(* IEC 61131-3 sources: test/Class/HmiMapFile, 1 file *)

(* ---- HmiMapFile.st ---- *)
(*!
<Class
	Name               = "HmiMapFile"
	Revision           = "0.0"
	RealtimeTask       = "false"
	CyclicTask         = "false"
	BackgroundTask     = "false"
	Sigmatek           = "true"
	OSInterface        = "false"
	HighPriority       = "false"
	Automatic          = "false"
	UpdateMode         = "Prescan"
	SharedCommandTable = "true"
	Objectsize         = "(284,120)">
	<Channels>
		<Server Name="ClassSvr" Visualized="false" Initialize="false" WriteProtected="true" Retentive="false"/>
		<Client Name="File" Required="true" Internal="false"/>
		<Client Name="StateBit" Required="true" Internal="false"/>
		<Client Name="StringLib" Required="true" Internal="false"/>
		<Client Name="VarList" Required="true" Internal="false"/>
	</Channels>
</Class>
*)
HmiMapFile : CLASS
  //Servers:
	ClassSvr 	: SvrChCmd_DINT;
  //Clients:
	File 	: CltChCmd_HmiFile;
	VarList 	: CltChCmd_HmiVarList;
	StateBit 	: CltChCmd_HmiStateBit35;
	StringLib 	: CltChCmd_HmiStrLib;
  //Variables:
		Tabs 	: DINT;
  //Functions:

	FUNCTION GLOBAL Create
		VAR_INPUT
			dp 	: ^CHAR;
			prjcrc 	: UDINT;
		END_VAR;

	FUNCTION GLOBAL TagLine
		VAR_INPUT
			ptxt 	: ^CHAR;
		END_VAR;

	FUNCTION GLOBAL TagNote
		VAR_INPUT
			ptag 	: ^CHAR;
		END_VAR;
  //Tables:
	FUNCTION @STD
		VAR_OUTPUT
			ret_code	: CONFSTATES;
		END_VAR;
	FUNCTION GLOBAL TAB @CT_;
END_CLASS;

#pragma usingLtd HmiFile
#pragma usingLtd HmiStateBit35
#pragma usingLtd HmiStrLib
#pragma usingLtd HmiVarList

FUNCTION GLOBAL HmiMapFile::TagLine
	VAR_INPUT
		ptxt 	: ^CHAR;
	END_VAR
  VAR
    tmp : array[0..10] of char;
  	dat : udint;
  END_VAR

  if(Tabs > 0) then
    _memset(#tmp[0], 9, sizeof(tmp));
    File.FWrite(#tmp[0], to_udint(Tabs));
  end_if;

  File.FWrite(ptxt, StringLib.StrLen(ptxt, 1));
  dat := 16#0A0D;
  File.FWrite(#dat, 2);

END_FUNCTION

FUNCTION GLOBAL HmiMapFile::TagNote
	VAR_INPUT
		ptag 	: ^char;
	END_VAR
  VAR
  	ph : ^char;
  END_VAR

  ph := ptag + 1;

  if(ph^ = '/') then
    Tabs -= 1;
  end_if;

  TagLine(ptag);

  if(ph^ <> '/') then
    Tabs += 1;
  end_if;

END_FUNCTION

FUNCTION GLOBAL HmiMapFile::Create
	VAR_INPUT
		dp 	: ^CHAR;
		prjcrc 	: UDINT;
	END_VAR
  VAR
    label : array[0..256] of char;
    idx : udint;
  END_VAR

(*
  crlf := 16#0A0D;

  StringLib.StrCpy(#label[0], 1, dp, 1);
  StringLib.StrCat(#label[0], 1, "EasyMap.txt", 1);

  File.FOpen(#label[0], 'W');

  StringLib.StrCpy(#label[0], 1, "[VER] := 2.0", 1);
  File.FWrite(#label[0], StringLib.StrLen(#label[0], 1));
  File.FWrite(#crlf, 2);

  StringLib.StrCpy(#label[0], 1, "[CRC] := 16#", 1);
  StringLib.HexToStr(#label[StringLib.StrLen(#label[0], 1)], prjcrc);
  File.FWrite(#label[0], StringLib.StrLen(#label[0], 1));
  File.FWrite(#crlf, 2);
  File.FWrite(#crlf, 2);

  idx := 0;
  while(VarList.GetMapInfo(idx, #label[0]) <> nil) do
    File.FWrite(#label[0], StringLib.StrLen(#label[0], 1));
    File.FWrite(#crlf, 2);
    idx += 1;
  end_while;
  File.FClose();
*)
  Tabs := 0;

  StringLib.StrCpy(#label[0], 1, dp, 1);
  StringLib.StrCat(#label[0], 1, "EasyMap.xml", 1);

  File.FOpen(#label[0], 'W');

  StringLib.StrCpy(#label[0], 1, "<?xml version=_1.0_ encoding=_ISO-8859-1_?>", 1);
  StringLib.StrXchg(#label[0], '_', '"');
  TagLine(#label[0]);

  TagNote("<mapinfo>");
    TagNote("<header>");
      StringLib.StrCpy(#label[0], 1, "<version value=_2.0_/>", 1);
      StringLib.StrXchg(#label[0], '_', '"');
      TagLine(#label[0]);

      StringLib.StrCpy(#label[0], 1, "<crc value=_0x", 1);
      StringLib.HexToStr(#label[StringLib.StrLen(#label[0], 1)], prjcrc);
      StringLib.StrCat(#label[0], 1, "_/>", 1);
      StringLib.StrXchg(#label[0], '_', '"');
      TagLine(#label[0]);
    TagNote("</header>");

    TagNote("<info>");
      idx := 0;
      while(VarList.GetMapInfoXML(idx, #label[0]) <> nil) do
        TagLine(#label[0]);
        idx += 1;
      end_while;

      idx := 0;
      while(StateBit.GetMapInfoXML(idx, #label[0]) <> nil) do
        TagLine(#label[0]);
        idx += 1;
      end_while;
    TagNote("</info>");
  TagNote("</mapinfo>");

  File.FClose();

END_FUNCTION
